(* CODESYS project AstroBROT.library
   Title: AstroBROT
   Version: 0.1
   Placeholder: AstroBROT
   Company: BROT

Project tree, tasks and I/O mapping:
  libraries: Tc2_Math, * (Beckhoff Automation GmbH); Tc2_Standard, * (Beckhoff Automation GmbH); Tc2_System, * (Beckhoff Automation GmbH); Tc2_Utilities, * (Beckhoff Automation GmbH); Tc3_Module, * (Beckhoff Automation GmbH); TcUnit, 1.2.0.0 (www.tcunit.org)
  Coordinates/
    function block CO_ABERRATION [ST]
    function block CO_REFRACT [ST]
    function CO_REFRACT_FORWARD [ST]
    function block FB_ALTAZ2HADEC [ST]
    function block FB_CO_NUTATE [ST]
    function block FB_Eq2Hor [ST]
    function block FB_Hor2Eq [ST]
    function block FB_NUTATE [ST]
    function block FB_PRECESS [ST]
    function block FB_SUNPOS [ST]
    data type S_EarthLocation
    data type S_SkyCoordEquatorial
    data type S_SkyCoordHorizontal
  Misc/
    function ATAN2 [ST]
    function Deg2Rad [ST]
    program MAIN [ST]
    function Rad2Deg [ST]
  Test/
    function block FB_DateTime2JD_Test [ST]
    function block FB_Eq2Hor_Test [ST]
    function block FB_JD2LST [ST]
  Time/
    function DateTime2JD [ST]
    function JD2LST [ST]
*)

// Coordinates/S_EarthLocation
TYPE S_EarthLocation :
STRUCT
	longitude:	LREAL;
	latitude:	LREAL;
	height:		LREAL;
END_STRUCT
END_TYPE

// Coordinates/S_SkyCoordEquatorial
TYPE S_SkyCoordEquatorial :
STRUCT
	ra:		LREAL;
	dec:	LREAL;
END_STRUCT
END_TYPE

// Coordinates/S_SkyCoordHorizontal
TYPE S_SkyCoordHorizontal :
STRUCT
	alt:	LREAL;
	az:		LREAL;
END_STRUCT
END_TYPE

// Coordinates/CO_ABERRATION
FUNCTION_BLOCK CO_ABERRATION
VAR_INPUT
	jd, 				// Julian Date
	ra, dec: LREAL; 	//ra and dec in degrees
	eps : LREAL := 0.0;
END_VAR
VAR_OUTPUT
	d_ra, d_dec: LREAL;
END_VAR
VAR
	sunpos: FB_SUNPOS;
	nutate: FB_NUTATE;
	sunra, sundec, sunlon,
	d_psi, d_epsilon, eps0,
	t, e, peri, cd, sd, ce, te, cp, sp, cs, ss, ca, sa, term1, term2, term3, term4: LREAL;
END_VAR
VAR CONSTANT
	d2r : LREAL := PI/180.0;
	k: LREAL := 20.49552; //constant of aberration, in arcseconds
	
END_VAR

(*
;+
;  NAME:
;     CO_ABERRATION
; PURPOSE:
;     Calculate changes to Ra and Dec due to the effect of annual aberration 
; EXPLANATION:
;      as described in Meeus, Chap 23.
; CALLING SEQUENCE:
;      co_aberration, jd, ra, dec, d_ra, d_dec, [EPS = ]
; INPUTS
;       jd      : Julian Date [scalar or vector]
;       ra, dec : Arrays (or scalars) of the ra  and dec's in degrees
;   Note: if jd is a vector, then ra and dec must either be scalars, or 
;                vectors of the same length.
;
; OUTPUTS
;       d_ra, d_dec: the corrections to ra and dec due to aberration in 
;                    arcseconds.  (These values can be added to the true RA 
;                    and dec to get the apparent position).   Note that d_ra
;                     is *not* multiplied by cos(dec), so that 
;                     apparent_ra = ra + d_ra/3600. 
; OPTIONAL INPUT KEYWORD:
;       eps : set this to the true obliquity of the ecliptic (in radians), or
;         it will be set for you if you don't know it (in that case, set it to
;                 an empty variable).
; EXAMPLE:
;   Compute the change in RA and Dec of Theta Persei (RA = 2h46m,11.331s, Dec =
;   49d20',54.54") due to aberration on 2028 Nov 13.19 TD
;
;      IDL> jdcnv,2028,11,13,.19*24,jd      ;Get Julian date
;      IDL> co_aberration,jd,ten(2,46,11.331)*15,ten(49,20,54.54),d_ra,d_dec
;
;      ==> d_ra = 30.045" (=2.003s)    d_dec = 6.697"
; NOTES:
;  These formula are from Meeus, Chapters 23.  Accuracy is much better than 1 
;   arcsecond.
;
;   The maximum deviation due to annual aberration is 20.49" and occurs when the
;   Earth velocity is perpendicular to the direction of the star.
;
; REVISION HISTORY:
;   Written, June 2002,      Chris O'Dell, U. of Wisconsin
;   Fix error with vector input   W. Landsman   June 2009
;   June 2009 update fixed case where JD was scalar but RA,Dec were vectors, but 
;     broke the case when both JD and RA,Dec were vectors Aug 2012 W. Landsman
;   Further fix when JD is 1 element vector  W. Landsman
;-
*)

T := (jd -2451545.0)/36525.0; // julian centuries from J2000 of jd.

IF EPS = 0.0 THEN
	// must calculate obliquity of ecliptic
	nutate(jd := jd, nut_long => d_psi, nut_obliq => d_epsilon); //d_psi and d_epsilon in degrees
	eps0 := ten(23,26,21.448)*3600.0 - 46.8150*T - 0.00059*EXPT(T, 2) +  0.001813*EXPT(T, 3);
	// TRUE obliquity OF the ecliptic in radians
	eps := (eps0 + d_epsilon)/3600.0*d2r; 	
END_IF

sunpos( JD := jd, RA => sunra, Dec => sundec, longmed => sunlon);

// Earth's orbital eccentricity
e := 0.016708634 - 0.000042037*T - 0.0000001267*EXPT(T, 2);
// longitude of perihelion, in degrees 
peri := 102.93735 + 1.71946*T + 0.00046*EXPT(T, 2);

//Useful Trig Functions
cd := COS(dec*d2r);		sd := SIN(dec*d2r);
ce := COS(eps); 		te := TAN(eps);
cp := COS(peri*d2r);	sp := SIN(peri*d2r);
cs := COS(sunlon*d2r);	ss := SIN(sunlon*d2r);
ca := COS(ra*d2r);		sa := SIN(ra*d2r);

term1 := (ca*cs*ce + sa*ss)/cd;
term2 := (ca*cp*ce + sa*sp)/cd;
term3 := (cs*ce*(te*cd - sa*sd) + ca*sd*ss);
term4 := (cp*ce*(te*cd - sa*sd) + ca*sd*sp);

d_ra := -k * term1 + e*k * term2;
d_dec := -k * term3 + e*k * term4;

END_FUNCTION_BLOCK

// Coordinates/FB_SUNPOS
FUNCTION_BLOCK FB_SUNPOS
VAR_INPUT
	// Julian Date
	JD:		LREAL;
	// output in Radians instead of Degrees
	RADIAN:	BOOL:= FALSE;
END_VAR
VAR_OUTPUT
	// right ascension
	RA,
	// declination of the sun
	Dec,
	// longitude
	longmed,
	// True Obliquity
	oblt:	LREAL;
END_VAR
VAR
	t, //  Julian centuries FROM 1900.0
	l, //  sun's mean longitude
	me, // Earth's mean anomaly
	ellcor, // ellipticity of the orbit
	mv, // mean anomaly of Venus
	vencorr,
	mm, 
	marscorr,
mj, jupcorr,
d, longterm, mooncorr,  omega:	LREAL;
END_VAR
VAR CONSTANT
	dtor: LREAL := PI/180.0; // Pi/180
END_VAR

(* source: https://idlastro.gsfc.nasa.gov/ftp/pro/astro/sunpos.pro *)

//  form TIME in Julian centuries FROM 1900.0
t := (jd - 2415020.0)/36525.0;

//  form sun's mean longitude
l := (279.696678+LMOD(36000.768925*t, 360.0))*3600.0;

//  allow for ellipticity of the orbit (equation of centre) using the Earth's mean anomaly ME
me := 358.475844 + LMOD(35999.049750*t, 360.0);
ellcor  := (6910.1 - 17.2*t)*SIN(me*dtor) + 72.3*SIN(2.0*me*dtor);
l := l + ellcor;
 
// allow FOR the Venus perturbations using the mean anomaly OF Venus MV
mv := 212.603219 + LMOD(58517.803875*t, 360.0);
vencorr := 4.8 * COS((299.1017 + mv - me)*dtor) + 
          5.5 * COS((148.3133 +  2.0 * mv  -  2.0 * me )*dtor) + 
          2.5 * COS((315.9433 +  2.0 * mv  -  3.0 * me )*dtor) + 
          1.6 * COS((345.2533 +  3.0 * mv  -  4.0 * me )*dtor) + 
          1.0 * COS((318.15   +  3.0 * mv  -  5.0 * me )*dtor);
l := l + vencorr;

//  Allow FOR the Mars perturbations using the mean anomaly OF Mars MM
mm := 319.529425  +  LMOD( 19139.858500 * t,  360.0 );
marscorr := 2.0 * COS((343.8883 -  2.0 * mm  +  2.0 * me)*dtor ) + 
            1.8 * COS((200.4017 -  2.0 * mm  + me) * dtor);
l := l + marscorr;

// Allow FOR the Jupiter perturbations using the mean anomaly OF Jupiter MJ
mj := 225.328328  +  LMOD( 3034.6920239 * t,  360.0 );
jupcorr := 7.2 * COS(( 179.5317 - mj + me )*dtor) + 
          2.6 * COS((263.2167  -  MJ ) *dtor) + 
          2.7 * COS(( 87.1450  -  2.0 * mj  +  2.0 * me ) *dtor) + 
          1.6 * COS((109.4933  -  2.0 * mj  +  me ) *dtor);
l := l + jupcorr;

// Allow FOR the Moons perturbations using the mean elongation OF the Moon from the Sun D
d := 350.7376814  + LMOD( 445267.11422 * t,  360.0 );
mooncorr  := 6.5 * SIN(d*dtor);
l := l + mooncorr;

// Allow for long period terms
longterm := 6.4 * SIN(( 231.19  +  20.20 * t )*dtor);
l :=  l + longterm;
l :=  LMOD( l + 2592000.0,  1296000.0); 
longmed := l/3600.0;

// Allow for Aberration
l :=  l - 20.5;

// Allow for Nutation using the longitude of the Moons mean node OMEGA
omega := 259.183275 - LMOD( 1934.142008 * t, 360.0);
l :=  l - 17.2 * SIN(omega*dtor);

// Form the True Obliquity
oblt := 23.452294 - 0.0130125*t + (9.2*COS(omega*dtor))/3600.0;

// Form Right Ascension AND Declination
l := l/3600.0;
ra := ATAN2( COS(l*dtor), SIN(l*dtor) * COS(oblt*dtor));
ra := MODABS(ra, 360.0);
dec := ASIN(SIN(l*dtor) * SIN(oblt*dtor));
 
IF RADIAN THEN
	oblt := oblt*dtor; 
	longmed := longmed*dtor;
ELSE
	ra := ra/dtor;
    dec := dec/dtor;
END_IF

END_FUNCTION_BLOCK

// Misc/ATAN2
FUNCTION ATAN2 : LREAL
VAR_INPUT
	y, x: LREAL;
END_VAR
VAR
END_VAR

(* source: https://de.wikipedia.org/wiki/Arctan2 *)
ATAN2 := 0.0;

IF x > 0 THEN
	ATAN2 := ATAN(y/x);
ELSIF x < 0 AND y > 0 THEN
	ATAN2 := ATAN(y/x) + PI;
ELSIF x < 0 AND y = 0 THEN
	ATAN2 := PI;
ELSIF x < 0 AND y < 0 THEN
	ATAN2 := ATAN(y/x) - PI;
ELSIF x = 0 AND y > 0 THEN
	ATAN2 := PI/2.0;
ELSIF x = 0 AND y < 0 THEN
	ATAN2 := -PI/2.0;
END_IF

END_FUNCTION

// Coordinates/FB_NUTATE
FUNCTION_BLOCK FB_NUTATE
VAR_INPUT
	jd:	LREAL;
END_VAR
VAR_OUTPUT
	nut_long, nut_obliq: LREAL := 0.0;
END_VAR
VAR
	t: LREAL;
	d, M, Mprime, F, omega: LREAL;
	arg, sarg, carg:  ARRAY[0..62] OF LREAL;
	I: INT;
END_VAR
VAR CONSTANT
	dtor:	LREAL := PI/180.0;
	coeff1:	ARRAY[0..3] OF LREAL := [297.85036, 445267.111480, -0.0019142,  1.0/189474];
	coeff2:	ARRAY[0..3] OF LREAL := [357.52772,  35999.050340, -0.0001603, -1.0/3E5]; 
	coeff3:	ARRAY[0..3] OF LREAL := [134.96298, 477198.867398,  0.0086972,  1.0/5.625E4]; 
	coeff4:	ARRAY[0..3] OF LREAL :=  [93.27191, 483202.017538, -0.0036825, -1.0/3.27270E5]; 
  	coeff5: ARRAY[0..3] OF LREAL := [125.04452,  -1934.136261,  0.0020708,  1.0/4.5E5];
	d_lng: ARRAY[0..62] OF LREAL := [0,-2,0,0,0,0,-2,0,0,-2,-2,-2,0,2,0,2,0,0,-2,0,2,0,0,-2,0,-2,0,0,2,-2,0,-2,0,0,2,2,0,-2,0,2,2,-2,-2,2,2,0,-2,-2,0,-2,-2,0,-1,-2,1,0,0,-1,0,0,2,0,2]; 
	m_lng: ARRAY[0..62] OF LREAL := [0,0,0,0,1,0,1,0,0,-1,17(0),2,0,2,1,0,-1,0,0,0,1,1,-1,0,0,0,0,0,0,-1,-1,0,0,0,1,0,0,1,0,0,0,-1,1,-1,-1,0,-1];
	mp_lng: ARRAY[0..62] OF LREAL := [0,0,0,0,0,1,0,0,1,0,1,0,-1,0,1,-1,-1,1,2,-2,0,2,2,1,0,0,-1,0,-1,0,0,1,0,2,-1,1,0,1,0,0,1,2,1,-2,0,1,0,0,2,2,0,1,1,0,0,1,-2,1,1,1,-1,3,0];
	f_lng: ARRAY[0..62] OF LREAL := [0,2,2,0,0,0,2,2,2,2,0,2,2,0,0,2,0,2,0,2,2,2,0,2,2,2,2,0,0,2,0,0,0,-2,2,2,2,0,2,2,0,2,2,0,0,0,2,0,2,0,2,-2,0,0,0,2,2,0,0,2,2,2,2];
	om_lng: ARRAY[0..62] OF LREAL := [1,2,2,2,0,0,2,1,2,2,0,1,2,0,1,2,1,1,0,1,2,2,0,2,0,0,1,0,1,2,1,1,1,0,1,2,2,0,2,1,0,2,1,1,1,0,1,1,1,1,1,0,0,0,0,0,2,0,0,2,2,2,2];
	sin_lng: ARRAY[0..62] OF LREAL := [-171996, -13187, -2274, 2062, 1426, 712, -517, -386, -301, 217, -158, 129, 123, 63, 63, -59, -58, -51, 48, 46, -38, -31, 29, 29, 26, -22, 21, 17, 16, -16, -15, -13, -12, 11, -10, -8, 7, -7, -7, -7, 6,6,6,-6,-6,5,-5,-5,-5,4,4,4,-4,-4,-4,3,-3,-3,-3,-3,-3,-3,-3 ];
	sdelt: ARRAY[0..62] OF LREAL := [-174.2, -1.6, -0.2, 0.2, -3.4, 0.1, 1.2, -0.4, 0, -0.5, 0, 0.1, 0,0,0.1, 0,-0.1,10(0), -0.1, 0, 0.1, 33(0)];
	cos_lng: ARRAY[0..62] OF LREAL := [ 92025, 5736, 977, -895, 54, -7, 224, 200, 129, -95,0,-70,-53,0, -33, 26, 32, 27, 0, -24, 16,13,0,-12,0,0,-10,0,-8,7,9,7,6,0,5,3,-3,0,3,3, 0,-3,-3,3,3,0,3,3,3, 14(0)] ;
	cdelt: ARRAY[0..62] OF LREAL := [8.9, -3.1, -0.5, 0.5, -0.1, 0.0, -0.6, 0.0, -0.1, 0.3, 53(0)];
END_VAR

//  form time in Julian centuries from 1900.0

t := (jd - 2451545.0)/36525.0;

// Mean elongation of the Moon

d := poly(T, coeff1)*dtor;
d := MODABS(d, 2.0*PI);

// Sun's mean anomaly

M := poly(T,coeff2)*dtor;
M := MODABS(M, 2.0*PI);

// Moon's mean anomaly

Mprime := poly(T,coeff3)*dtor;
Mprime := MODABS(Mprime, 2.0*PI);

// Moon's argument of latitude

F := poly(T, coeff4 )*dtor;
F := MODABS(F, 2.0*PI);

// Longitude OF the ascending node OF the Moon's mean orbit on the ecliptic,
//  measured from the mean equinox of the date

omega := poly(T, coeff5)*dtor;
omega := MODABS(omega, 2.0*PI);


// Sum the periodic terms 
FOR i:=0 TO 62 DO
	arg[i] := d_lng[i]*d + m_lng[i]*m +mp_lng[i]*mprime + f_lng[i]*f +om_lng[i]*omega;
	sarg[i] := SIN(arg[i]);
	carg[i] := COS(arg[i]);
END_FOR

nut_long  := 0.0;
nut_obliq := 0.0;

FOR i:=0 TO 62 DO
	nut_long  := nut_long  + 0.0001*( (sdelt[i]*t + sin_lng[i])*sarg[i]);
	nut_obliq := nut_obliq + 0.0001*( (cdelt[i]*t + cos_lng[i])*carg[i]);
END_FOR

END_FUNCTION_BLOCK

// Coordinates/CO_REFRACT
FUNCTION_BLOCK CO_REFRACT
VAR_INPUT
	old_alt: 		LREAL;
	height: 		LREAL;
	altitude: 		LREAL := 0.0;
	pressure: 		LREAL := 0.0;
	temperature: 	LREAL := 0.0;
	epsilon: 		LREAL := 0.25; //accuracy of iteration for observed=TRUE case, in arcseconds
	TO_OBSERVED: 	BOOL;
END_VAR
VAR_OUTPUT
	new_alt: 		LREAL;
END_VAR
VAR
	aout, P, T, dr, cur, last : LREAL;
END_VAR
VAR CONSTANT
	alpha : LREAL := 0.0065; //temp lapse rate [deg C per meter]
END_VAR

// based on IDLAstro's co_refract
// https://github.com/wlandsman/IDLAstro/blob/master/pro/co_refract.pro

// estimate a temperature, if None is given
IF temperature = 0.0 THEN
	IF height > 11000.0 THEN 
		temperature := 211.5; 
	ELSE 
		temperature := 283.0 - alpha * height;
	END_IF
END_IF

// estimate Pressure based on altitude, using U.S. Standard Atmosphere formula.
IF pressure = 0 THEN 
	pressure := 1010.0 * EXPT(1 - 6.5 / 288000 * height, 5.255);
END_IF

IF NOT TO_OBSERVED THEN 
	aout := old_alt - co_refract_forward(old_alt, pressure:=pressure,temperature:=temperature);
ELSE
	aout := 0.0;
	P := pressure; 
	T := temperature;
	//calculate initial refraction guess
	dr := co_refract_forward(old_alt, pressure:=P, temperature:=T);
	cur := old_alt + dr; // guess of observed location

	REPEAT 
	 	last := cur;
		dr := co_refract_forward(cur, pressure:= P, temperature:=T);
	  	cur := old_alt + dr;
	UNTIL ABS(last-cur)*3600.0 < epsilon
	END_REPEAT
	aout := cur;
END_IF

new_alt := aout;

END_FUNCTION_BLOCK

// Coordinates/CO_REFRACT_FORWARD
FUNCTION CO_REFRACT_FORWARD : LREAL
VAR_INPUT
	// The observed (apparent) altitude, in DEGREES.
	altitude: 		LREAL;
	// Pressure [in millibars]. Default is 1010 millibars.
	pressure: 		LREAL := 1010.0;
	// Ground Temp [in Celsius].  Default is 0 Celsius.
	temperature: 	LREAL := 0.0;
END_VAR
VAR
	Ref:			LREAL;
	tpcor: 			LREAL;
END_VAR
VAR CONSTANT
	d2r : LREAL := PI/180.0;
END_VAR

// based on IDLAstro's co_refract_forward
// https://github.com/wlandsman/IDLAstro/blob/master/pro/co_refract.pro

// limit values to reasonable ranges
altitude := LIMIT(0.0, altitude, 90.0);
pressure := LIMIT(600.0, pressure, 1200.0);
temperature := LIMIT(-40.0, temperature, 40.0);

// calculate refraction depending on altitude
IF altitude >= 15.0 THEN
	Ref := 1.0 / TAN(Deg2Rad(altitude + 7.31/(altitude + 4.4)));
ELSE
	Ref := 3.569*(0.1594 + 0.0196*altitude + 0.00002*EXPT(altitude, 2))/(1.0+0.505*altitude + 0.0845*EXPT(altitude, 2));
END_IF

// correct and return
tpcor := pressure * 283.15 / (1010.0 * (273.15 + temperature));
CO_REFRACT_FORWARD := tpcor * Ref;

END_FUNCTION

// Misc/Deg2Rad
FUNCTION Deg2Rad : LREAL
VAR_INPUT
	deg: LREAL;
END_VAR
VAR
END_VAR

Deg2Rad := deg / 180.0 * PI;

END_FUNCTION

// Coordinates/FB_ALTAZ2HADEC
FUNCTION_BLOCK FB_ALTAZ2HADEC
VAR_INPUT
	// the local apparent altitude, in DEGREES
	alt:	LREAL;
	// the local apparent azimuth, in DEGREES
	az:		LREAL;
	// the local geodetic latitude, in DEGREES
	lat: 	LREAL;
END_VAR
VAR_OUTPUT
	// the local apparent hour angle, in DEGREES
	ha:		LREAL;
	// the local apparent declination, in DEGREES
	dec:	LREAL;
END_VAR
VAR
	alt_r:	LREAL;
	az_r:	LREAL;
	lat_r:	LREAL;
	sindec: LREAL;
END_VAR
VAR CONSTANT
	d2r:	LREAL := PI/180.0;
	//r2d:	LREAL := 180.0/PI;
	//h2r:	LREAL := PI/12.0;
	//h2d:	LREAL := 15.0;
END_VAR

(*

  NAME:
    ALTAZ2HADEC
 PURPOSE:
    Convert Horizon (Alt-Az) coordinates to Hour Angle and Declination.
 EXPLANATION::
    Can deal with the NCP singularity.    Intended mainly to be used by
    program hor2eq.pro
 CALLING SEQUENCE:
   ALTAZ2HADEC, alt, az, lat, ha, dec

 INPUTS
   alt - the local apparent altitude, in DEGREES, scalar or vector
   az  - the local apparent azimuth, in DEGREES, scalar or vector,
         measured EAST of NORTH!!!  If you have measured azimuth west-of-south
        (like the book MEEUS does), convert it to east of north via:
                       az = (az + 180) mod 360

   lat -  the local geodetic latitude, in DEGREES, scalar or vector.

 OUTPUTS
   ha  -  the local apparent hour angle, in DEGREES.  The hour angle is the 
          time that right ascension of 0 hours crosses the local meridian.  
          It is unambiguously defined.
   dec -  the local apparent declination, in DEGREES.

 EXAMPLE:
     Arcturus is observed at an apparent altitude of 59d,05m,10s and an 
     azimuth (measured east of north) of 133d,18m,29s while at the 
     latitude of +43.07833 degrees.
     What are the local hour angle and declination of this object?

     IDL> altaz2hadec, ten(59,05,10), ten(133,18,29), 43.07833, ha, dec
     ===> Hour angle ha = 336.683 degrees
          Declination, dec = 19.1824 degrees

       The widely available XEPHEM code gets:
                 Hour Angle = 336.683
                 Declination = 19.1824

 REVISION HISTORY:
    Written  Chris O'Dell Univ. of Wisconsin-Madison May 2002
*)
alt_r  := alt*d2r;
az_r := az*d2r;
lat_r := lat*d2r;

//******************************************************************************
// find local HOUR ANGLE (in degrees, from 0. to 360.)
ha := atan2( -SIN(az_r)*COS(alt_r), 
           -COS(az_r)*SIN(lat_r)*COS(alt_r)+SIN(alt_r)*COS(lat_r));
ha := ha / d2r;
IF ha < 0.0 THEN 
	ha := ha + 360.0;
END_IF
 ha := MODABS(ha, 360.0);

// Find declination (positive if north of Celestial Equator, negative if south)
sindec := SIN(lat_r)*SIN(alt_r) + COS(lat_r)*COS(alt_r)*COS(az_r);
// convert dec to degrees
dec := ASIN(sindec)/d2r;

END_FUNCTION_BLOCK

// Coordinates/FB_CO_NUTATE
FUNCTION_BLOCK FB_CO_NUTATE
VAR_INPUT
	jd,
	ra,
	dec:	LREAL;
END_VAR
VAR_OUTPUT
	d_ra,
	d_dec,
	eps,
	d_psi,
	d_eps:	LREAL;
END_VAR
VAR
	T, 
	eps0,
ce, se,x,y,z,x2,y2,z2,rad,xyproj,ra2,dec2: LREAL;
	nutate:	FB_NUTATE;
END_VAR
VAR CONSTANT
	d2r:	LREAL := PI/180.0;
	d2as:	LREAL := PI/(180.0*3600.0);
END_VAR

// Julian centuries FROM J2000 OF jd.
T := (jd -2451545.0)/36525.0; 

// must calculate obliquity OF ecliptic
nutate(jd := jd,
		nut_long => d_psi, 
		nut_obliq => d_eps); 

eps0 := 23.4392911*3600.0 - 46.8150*T - 0.00059*EXPT(T, 2) + 0.001813*EXPT(T, 3);
eps := (eps0 + d_eps)/3600.0*d2r; // TRUE obliquity OF the ecliptic in radians
 
//useful numbers
ce := COS(eps);
se := SIN(eps);

// convert ra-dec to equatorial rectangular coordinates
x := COS(ra*d2r) * COS(dec*d2r);
y := SIN(ra*d2r) * COS(dec*d2r);
z := SIN(dec*d2r);

// apply corrections to each rectangular coordinate
x2 := x - (y*ce + z*se)*d_psi * d2as;
y2 := y + (x*ce*d_psi - z*d_eps) * d2as;
z2 := z + (x*se*d_psi + y*d_eps) * d2as;

// convert back to equatorial spherical coordinates
rad := SQRT(x2*x2 + y2*y2 + z2*z2);
xyproj := SQRT(x2*x2 + y2*y2);

ra2  := x2 * 0.0;
dec2 := x2 * 0.0;

// Calculate Ra and Dec in RADIANS (later convert to DEGREES)
IF (xyproj = 0) AND (z <> 0) THEN
	// places where xyproj=0 (point at NCP or SCP)
	dec2 := ASIN(z2/rad);
	ra2 := 0.0;
END_IF
 
IF (xyproj <> 0) THEN
	// places other than NCP or SCP
	ra2 := ATAN2(y2, x2);
	dec2 := ASIN(z2/rad);
END_IF

// convert to DEGREES

ra2 := ra2 /d2r;
dec2 := dec2 /d2r;

ra2 := MODABS(ra2, 360.0);


// Return changes in ra and dec in arcseconds
d_ra := (ra2 - ra) * 3600.0;
d_dec := (dec2 - dec) * 3600.0;

END_FUNCTION_BLOCK

// Coordinates/FB_Eq2Hor
FUNCTION_BLOCK FB_Eq2Hor
VAR_INPUT
	in_coord:	S_SkyCoordEquatorial;
	JD:         LREAL;
	location:   S_EarthLocation;
END_VAR
VAR_OUTPUT
	out_coord:	S_SkyCoordHorizontal;
END_VAR
VAR
	lst:		LREAL;
	ha:			LREAL;
	_dec: 		LREAL;
	_lat:		LREAL;
	_ha:		LREAL;
	_alt:		LREAL;
	_az:		LREAL;
END_VAR
VAR CONSTANT
END_VAR

// following "Practical astronomy with your calculator" by Peter Duffett-Smith

// calculate hour angle in degrees
lst := JD2LST(JD := JD, loc := location);
ha := lst - in_coord.ra;

// to rad
_dec := Deg2Rad(in_coord.dec);
_lat := Deg2Rad(location.latitude);
_ha  := Deg2Rad(ha);

// find alt
_alt := ASIN(SIN(_dec) * SIN(_lat) + COS(_dec) * COS(_lat) * COS(_ha));
out_coord.alt := Rad2Deg(_alt);

// find az
_az := ACOS((SIN(_dec) - SIN(_lat) * SIN(_alt)) / (COS(_lat) * COS(_alt)));
out_coord.az := Rad2Deg(_az);

// if sin(ha) is positive, calculate true azimuth
IF SIN(_ha) > 0 THEN
	out_coord.az := 360.0 - out_coord.az;
END_IF

END_FUNCTION_BLOCK

// Time/JD2LST
FUNCTION JD2LST : LREAL
VAR_INPUT
	JD: 	LREAL;
	loc:	S_EarthLocation;
END_VAR
VAR
	T: 		LREAL;
	theta0: LREAL;
	gmst:	LREAL;
END_VAR

// following https://squarewidget.com/astronomical-calculations-sidereal-time/
T := ((JD - 2451545.0) / 36525.0);
theta0 := 280.46061837 + 360.98564736629 * (JD - 2451545.0) + (0.000387933 * T * T) - (T * T * T / 38710000.0); // (12.4)
gmst := MODABS(theta0, 360.0);
JD2LST := gmst + loc.longitude; // LST in degrees

END_FUNCTION

// Misc/Rad2Deg
FUNCTION Rad2Deg : LREAL
VAR_INPUT
	rad: LREAL;
END_VAR
VAR
END_VAR

Rad2Deg := rad / PI * 180.0;

END_FUNCTION

// Coordinates/FB_Hor2Eq
FUNCTION_BLOCK FB_Hor2Eq
VAR_INPUT
	in_coord: 	S_SkyCoordHorizontal;
	JD: 		LREAL;
	location:	S_EarthLocation;
	out_coord:	S_SkyCoordEquatorial;

	precess:	BOOL := TRUE;
	NUTATE:		BOOL := TRUE;
	aberration:	BOOL := TRUE;
	refract:	BOOL := TRUE;
	altitude:	LREAL := 0.0;
END_VAR
VAR_OUTPUT
	// Right Ascension of object  (J2000) in degrees (FK5)
	ra: 	LREAL;
	// Declination of object (J2000) in degrees (FK5)
	dec:	LREAL;
	// hour angle (in degrees) (optional)
	ha:		LREAL;
END_VAR
VAR
	
	alt_,
	az_,
	lmst,
	J_now: LREAL;
	co_nutate: 		FB_CO_NUTATE;
	co_aberration: 	CO_ABERRATION;
	co_refract:		CO_REFRACT;
	fbprecess:		FB_PRECESS;
	altaz2hadec:	FB_ALTAZ2HADEC;
	last: LREAL;
	dra1: LREAL;
	ddec1: LREAL;
	eps: LREAL;
	d_psi: LREAL;
	dra2: LREAL;
	ddec2: LREAL;
END_VAR
VAR CONSTANT
	//d2r:	LREAL := PI/180.0;
	//r2d:	LREAL := 180.0/PI;
	//h2r:	LREAL := PI/12.0;
	h2d:	LREAL := 15.0;
END_VAR

// store alt/az, so we don't change ra, dec arrays.
alt_ := in_coord.alt;   
az_ := in_coord.az;


// Make Correction for ATMOSPHERIC REFRACTION
// (use this for visible and radio wavelengths; author is unsure about other wavelengths)
IF refract THEN 
	co_refract(old_alt := alt_, 
			   altitude := altitude, 
			   to_observed := TRUE, 
			   new_alt => alt_);
END_IF

co_nutate(	jd := jd, 
			ra := 45.0, 
			dec := 45.0, 
			d_ra => dra1, 
			d_dec => ddec1, 
			eps => eps, 
			d_psi => d_psi);
//******************************************************************************
//Calculate LOCAL APPARENT SIDEREAL TIME
// first get local mean sidereal time (lmst)
// get LST (btw, THIS is the RA OF the zenith) 
// note:this is indep of tzone since giving jd
lmst := JD2LST(JD := JD, loc := location);

// calculate local APPARENT sidereal time (last)
// ADD correction in degrees
last := lmst + d_psi *COS(eps)/3600.0 ; 

//****************************************************************************
// Now do the spherical trig to get APPARENT Hour Angle [degrees], and
// declination [degrees].
altaz2hadec( alt := alt_, az := az_, lat := lat, ha => ha, dec => dec);

// Find Right Ascension (in degrees, from 0 to 360.)
 ra := MODABS(last - ha + 360.0, 360.0);



//*****************************************************************************
// calculate NUTATION and ABERRATION Corrections to Ra-Dec
IF NUTATE THEN
	co_nutate(	jd := jd, 
			ra := ra, 
			dec := dec, 
			d_ra => dra1, 
			d_dec => ddec1, 
			eps => eps, 
			d_psi => d_psi);
ELSE
	dra1 := 0.0;
	ddec1 := 0.0;	
END_IF
IF aberration THEN
	co_aberration(	jd := jd, 
				ra := ra, 
				dec := dec, 
				d_ra => dra2, 
				d_dec => ddec2, 
				eps := eps);
ELSE
	dra2 := 0.0;
	ddec2 := 0.0;	
END_IF
//******************************************************************************
// Make Nutation and Aberration Corrections (if wanted)

ra := ra - (dra1 + dra2)/3600.0;
dec := dec - (ddec1 + ddec2)/3600.0;
 //compute current equinox
J_now := (JD - 2451545.0)/365.25 + 2000.0 ;

//*****************************************************************************
// PRECESS coordinates to current date
// (uses astro lib procedure PRECESS.pro)

IF precess THEN 
	fbprecess( ra := ra, dec := dec, 
	EQUINOX1 := 2000.0, EQUINOX2 := J_now, 
	ra_precessed =>ra, dec_precessed => dec);                   
END_IF

// set output
out_coord.ra := ra;
out_coord.dec := dec;

END_FUNCTION_BLOCK

// Coordinates/FB_PRECESS
FUNCTION_BLOCK FB_PRECESS
VAR_INPUT
	ra, 
	dec,
	equinox1,
	equinox2: LREAL;
	RADIAN:	BOOL := FALSE;
END_VAR
VAR_OUTPUT
	ra_precessed,
	dec_precessed:	LREAL;
END_VAR
VAR
	ra_rad, dec_rad: LREAL;
	a,b,c,t: LREAL;
	x, x2: ARRAY[0..2] OF LREAL;
	st1: LREAL;
	rot: ARRAY[0..2,0..2] OF LREAL;
	sina, sinb, sinc, cosa,cosb,cosc: LREAL;
END_VAR
VAR CONSTANT
	deg_to_rad : LREAL := PI/180.0;
	sec_to_rad : LREAL := deg_to_rad/3600.0;
END_VAR

IF NOT RADIAN THEN
	ra_rad := ra*deg_to_rad;
	dec_rad := dec*deg_to_rad;
ELSE
    //Convert TO double precision IF NOT already
	ra_rad := ra;
	dec_rad := dec;
END_IF

a := COS( dec_rad );
x[0] := a*COS(ra_rad); x[1] := a*SIN(ra_rad); x[2] := SIN(dec_rad);

//*** PREMAT code starts here
ST1 := 0.001*( equinox1 - 2000.0);
t := 0.001*( equinox2 - equinox1);
//  Compute 3 rotation angles
A := sec_to_rad * T * (23062.181 + ST1*(139.656 +0.0139*ST1) + T*(30.188 - 0.344*ST1+17.998*T));
B := sec_to_rad * T * T * (79.280 + 0.410*ST1 + 0.205*T) + A;
C := sec_to_rad * T * (20043.109 - ST1*(85.33 + 0.217*ST1) + T*(-42.665 - 0.217*ST1 -41.833*T));
  sina := SIN(a); sinb := SIN(b);  sinc := SIN(c);
  cosa := COS(a); cosb := COS(b);  cosc := COS(c);

rot[0,0] :=  cosa*cosb*cosc-sina*sinb; 	rot[0,1] := sina*cosb+cosa*sinb*cosc; 	rot[0,2] := cosa*sinc;
rot[1,0] := -cosa*sinb-sina*cosb*cosc; 	rot[1,1] := cosa*cosb-sina*sinb*cosc; 	rot[1,2] := -sina*sinc;
rot[2,0] := -cosb*sinc;					rot[2,1] := -sinb*sinc; 				rot[2,2] := cosc;

//*** PREMAT code ends here

//x2 := rot* x; //rotate to get output direction cosines
x2[0] := rot[0,0]*x[0] + rot[1,0]*x[1] + rot[2,0]*x[2];
x2[1] := rot[0,1]*x[0] + rot[1,1]*x[1] + rot[2,1]*x[2];
x2[2] := rot[0,2]*x[0] + rot[1,2]*x[1] + rot[2,2]*x[2];

ra_rad := atan2(x2[1],x2[0]);
dec_rad := ASIN(x2[2]);

IF NOT RADIAN THEN
	ra_precessed := ra_rad/deg_to_rad;
	ra_precessed := MODABS(ra_precessed, 360.0);            //RA between 0 AND 360 degrees
	dec_precessed := dec_rad/deg_to_rad;
ELSE
	ra_precessed := ra_rad; 
	dec_precessed := dec_rad;
	ra_precessed := MODABS(ra_rad, 2.0*PI);
END_IF

END_FUNCTION_BLOCK

// Misc/MAIN
PROGRAM MAIN
VAR
	fbDateTime2JB : FB_DateTime2JD_Test;
	fbEq2Hor_Test : FB_Eq2Hor_Test;
	fbJD2LST_Test : FB_JD2LST;
END_VAR

TcUnit.RUN();

END_PROGRAM

// Test/FB_DateTime2JD_Test
FUNCTION_BLOCK FB_DateTime2JD_Test EXTENDS TcUnit.FB_TestSuite
VAR_INPUT
END_VAR
VAR_OUTPUT
END_VAR
VAR
	time1: TIMESTRUCT := (wYear := 2000, wMonth := 1, wDay := 1);
	output1: LREAL;
	jd1: LREAL := 2451544.50000;
	
	time2: TIMESTRUCT := (wYear := 2023, wMonth := 7, wDay := 17, wHour := 11, wMinute := 15, wSecond := 32);
	output2: LREAL;
	jd2: LREAL := 2460142.96912;
END_VAR

TEST('DateTime2JD');

output1 := DateTime2JD(time1);
AssertEquals_LREAL(Expected := jd1, Actual := output1, Delta := 1E-5, Message := 'Wrong JD1'); 

output2 := DateTime2JD(time2);
AssertEquals_LREAL(Expected := jd2, Actual := output2, Delta := 1E-5, Message := 'Wrong JD2'); 

TEST_FINISHED();

END_FUNCTION_BLOCK

// Time/DateTime2JD
FUNCTION DateTime2JD : LREAL
VAR_INPUT
	epoch: TIMESTRUCT;
END_VAR
VAR
	a,y,m,d,jdn: LREAL;
END_VAR

(*    import datetime
    from math import floor
    if not type(epoch) is datetime.datetime:
        raise TypeError('datetime must be of type datetime')
    
    a = floor((14 - epoch.month)/12)
    y = epoch.year + 4800 - a
    m = epoch.month + 12*a - 3
    
    d = epoch.day
    d += epoch.hour/24. + epoch.minute/1440. + epoch.second/86400. # microsecond might be added here?
    
    if [epoch.year,epoch.month,d] >= [1582,10,15]:
        jdn = epoch.day + floor((153*m + 2)/5) + 365*y + floor(y/4) - floor(y/100) + floor(y/400) - 32045
    elif [epoch.year,epoch.month,d] <= [1582,10,4]:
        jdn = epoch.day + floor((153*m + 2)/5) + 365*y + floor(y/4) - 32083
    return jdn + (epoch.hour-12)/24. + epoch.minute/1440. + epoch.second/86400.
*)
a := FLOOR((14.0 - epoch.wMonth)/12.0);
y := epoch.wYear + 4800.0 - a;
m := epoch.wMonth + 12.0*a - 3.0;

d := epoch.wDay + (epoch.wHour/24.0) + (epoch.wMinute/1440.0) + (epoch.wSecond/86400.0);

//IF (epoch.wYear > 1582) (* AND (epoch.wMonth > 10.0) AND (d > 15.0)*) THEN
	jdn := epoch.wDay + FLOOR((153*m + 2)/5) + 365.0*y + FLOOR(y/4) - FLOOR(y/100) + FLOOR(y/400) - 32045.0;
//ELSIF (epoch.wYear < 1582) AND (epoch.wMonth < 10) AND (d > 4.0) THEN
//	jdn := epoch.wDay + FLOOR((153*m + 2)/5) + 365.0*y + FLOOR(y/4) - 32083.0;
//END_IF

DateTime2JD := jdn
			+ (epoch.wHour-12.0)/24.0
			+ (epoch.wMinute/1440.0) 
			+ (epoch.wSecond/86400.0)
			+ (DWORD_TO_REAL(epoch.wMilliseconds)/86400000.0);

END_FUNCTION

// Test/FB_Eq2Hor_Test
FUNCTION_BLOCK FB_Eq2Hor_Test EXTENDS TcUnit.FB_TestSuite
VAR_INPUT
END_VAR
VAR_OUTPUT
END_VAR
VAR
	jd: LREAL := 2451544.50000; // 1/1/2000
	loc0: S_EarthLocation := (longitude := 0, latitude := 0, height := 0);
	loc1: S_EarthLocation := (longitude := 10, latitude := 52, height := 0);
	
	in_coord1: S_SkyCoordEquatorial := (ra := 0, dec := 0);
	out_coord1: S_SkyCoordHorizontal;
	exp_coord1: S_SkyCoordHorizontal := (alt := -9.9678, az := 270.0);
	
	in_coord2: S_SkyCoordEquatorial := (ra := 10.0 * 15.0, dec := 30);
	out_coord2: S_SkyCoordHorizontal;
	exp_coord2: S_SkyCoordHorizontal := (alt := 33.8001277, az := 53.0084778);
	
	in_coord3: S_SkyCoordEquatorial := (ra := 10.0 * 15.0, dec := 30);
	out_coord3: S_SkyCoordHorizontal;
	exp_coord3: S_SkyCoordHorizontal := (alt := 53.3456083, az := 111.0780528);
	
	eq2hor: FB_Eq2Hor;
END_VAR

TEST('0RaDec2AltAzAtLoc0');
eq2hor(in_coord:=in_coord1, JD:=jd, location:=loc0, out_coord=>out_coord1);
AssertEquals_LREAL(Expected := exp_coord1.alt, Actual := out_coord1.alt, Delta := 1E-5, Message := 'Alt conversion failed.');
AssertEquals_LREAL(Expected := exp_coord1.az, Actual := out_coord1.az, Delta := 1E-5, Message := 'Az conversion failed.');

TEST('RaDec2AltAzAtLoc0');
eq2hor(in_coord:=in_coord2, JD:=jd, location:=loc0, out_coord=>out_coord2);
AssertEquals_LREAL(Expected := exp_coord2.alt, Actual := out_coord2.alt, Delta := 1E-5, Message := 'Alt conversion failed.');
AssertEquals_LREAL(Expected := exp_coord2.az, Actual := out_coord2.az, Delta := 1E-5, Message := 'Az conversion failed.');

TEST('RaDec2AltAzAtLoc1');
eq2hor(in_coord:=in_coord3, JD:=jd, location:=loc1, out_coord=>out_coord3);
AssertEquals_LREAL(Expected := exp_coord3.alt, Actual := out_coord3.alt, Delta := 1E-5, Message := 'Alt conversion failed.');
AssertEquals_LREAL(Expected := exp_coord3.az, Actual := out_coord3.az, Delta := 1E-5, Message := 'Az conversion failed.');

TEST_FINISHED();

END_FUNCTION_BLOCK

// Test/FB_JD2LST
FUNCTION_BLOCK FB_JD2LST EXTENDS TcUnit.FB_TestSuite
VAR_INPUT
END_VAR
VAR_OUTPUT
END_VAR
VAR
	loc0: S_EarthLocation := (longitude := 0, latitude := 0, height := 0);
	loc1: S_EarthLocation := (longitude := 10, latitude := 52, height := 0);

	jd1: LREAL := 2451557.5;
	lst1: LREAL;
	exp1: LREAL := 112.7812104487;
	lst2: LREAL;
	exp2: LREAL := 122.7812104487;	
END_VAR

TEST('loc0');
lst1 := JD2LST(JD := jd1, loc := loc0);
AssertEquals_LREAL(Expected := exp1, Actual := lst1, Delta := 1E-5, Message := 'Wrong LST.');

TEST('loc1');
lst2 := JD2LST(JD := jd1, loc := loc1);
AssertEquals_LREAL(Expected := exp2, Actual := lst2, Delta := 1E-5, Message := 'Wrong LST.');

TEST_FINISHED();

END_FUNCTION_BLOCK
